// TIA Portal V17 export
// export: Created 2026-04-13T11:12:52.8832343Z, ExportSetting WithDefaults, DisplayName Totally Integrated Automation Portal, DisplayVersion V17 Update 4, DisplayName TIA Portal Openness, DisplayVersion V17 Update 4, DisplayName TIA Portal Version Control Interface, DisplayVersion V17, DisplayName SINAMICS Startdrive Advanced, DisplayVersion V17, DisplayName SINAMICS Startdrive G130, G150, S120, S150, SINAMICS MV, S210, DisplayVersion V17, DisplayName SINAMICS Startdrive G110M, G120, G120C, G120D, G120P, G115D, DisplayVersion V17, DisplayName STEP 7 Professional, DisplayVersion V17 Update 4, DisplayName STEP 7 Safety, DisplayVersion V17, DisplayName WinCC Professional, DisplayVersion V17 Update 4
TagTable "INCIP"
  INCIP_DD电导合格值 : Real  (PLC tag INCIP.DD电导合格值, HMI_连接_1, 1 s)
  INCIP_JX碱洗温度设定 : Real  (PLC tag INCIP.JX碱洗温度设定, HMI_连接_1, 1 s)
  INCIP_DD电导率当前值 : Real  (PLC tag INCIP.DD电导率当前值, HMI_连接_1, 1 s)
  INCIP_JX碱洗温度 : Real  (PLC tag INCIP.JX碱洗温度, HMI_连接_1, 1 s)
  INCIP_CIP压力 : Real  (PLC tag INCIP.CIP压力, HMI_连接_1, 1 s)
  INCIP_MZD自动清洗 : Bool  (PLC tag INCIP.MZD自动清洗, HMI_连接_1, 1 s)
  INCIP_MSD手动_纯水清洗 : Bool  (PLC tag INCIP.MSD手动_纯水清洗, HMI_连接_1, 1 s)
  INCIP_MSD手动_碱水清洗 : Bool  (PLC tag INCIP.MSD手动_碱水清洗, HMI_连接_1, 1 s)
  INCIP_MSD手动_溶剂清洗 : Bool  (PLC tag INCIP.MSD手动_溶剂清洗, HMI_连接_1, 1 s)
  INCIP_MSD手动_热水清洗 : Bool  (PLC tag INCIP.MSD手动_热水清洗, HMI_连接_1, 1 s)
  INCIP_MQX清洗重置 : Bool  (PLC tag INCIP.MQX清洗重置, HMI_连接_1, 1 s)
  INCIP_MCS纯水罐阀门 : Bool  (PLC tag INCIP.MCS纯水罐阀门, HMI_连接_1, 1 s)
  INCIP_MJS碱水罐阀门 : Bool  (PLC tag INCIP.MJS碱水罐阀门, HMI_连接_1, 1 s)
  INCIP_MZS注射水阀门 : Bool  (PLC tag INCIP.MZS注射水阀门, HMI_连接_1, 1 s)
  INCIP_MYK压空吹干阀 : Bool  (PLC tag INCIP.MYK压空吹干阀, HMI_连接_1, 1 s)
  INCIP_MD清洗失败 : Bool  (PLC tag INCIP.MD清洗失败, HMI_连接_1, 1 s)
  INCIP_MQX室内清洗辅助 : Bool  (PLC tag INCIP.MQX室内清洗辅助, HMI_连接_1, 1 s)
  INCIP_MZT主塔清洗头 : Bool  (PLC tag INCIP.MZT主塔清洗头, HMI_连接_1, 1 s)
  INCIP_MZT中途停止 : Bool  (PLC tag INCIP.MZT中途停止, HMI_连接_1, 1 s)
  INCIP_MXT心跳信号发送 : Bool  (PLC tag INCIP.MXT心跳信号发送, HMI_连接_1, 1 s)
  INCIP_MXT心跳信号接受 : Bool  (PLC tag INCIP.MXT心跳信号接受, HMI_连接_1, 1 s)
  INCIP_MXY泄压请求 : Bool  (PLC tag INCIP.MXY泄压请求, HMI_连接_1, 1 s)
  INCIP_MGS供水泵请求 : Bool  (PLC tag INCIP.MGS供水泵请求, HMI_连接_1, 1 s)
  INCIP_MCIP远程状态 : Bool  (PLC tag INCIP.MCIP远程状态, HMI_连接_1, 1 s)
  INCIP_QCS纯水罐阀门 : Bool  (PLC tag INCIP.QCS纯水罐阀门, HMI_连接_1, 1 s)
  INCIP_QJS碱水罐阀门 : Bool  (PLC tag INCIP.QJS碱水罐阀门, HMI_连接_1, 1 s)
  INCIP_QZS注射水罐阀门 : Bool  (PLC tag INCIP.QZS注射水罐阀门, HMI_连接_1, 1 s)
  INCIP_QYG压干阀门 : Bool  (PLC tag INCIP.QYG压干阀门, HMI_连接_1, 1 s)
  INCIP_QGS供水泵状态CIP : Bool  (PLC tag INCIP.QGS供水泵状态CIP, HMI_连接_1, 1 s)
  INCIP_QXY泄压阀门 : Bool  (PLC tag INCIP.QXY泄压阀门, HMI_连接_1, 1 s)
  INCIP_PS排水时间 : Real  (PLC tag INCIP.PS排水时间, HMI_连接_1, 1 s)
  INCIP_PS排水时间计时 : Real  (PLC tag INCIP.PS排水时间计时, HMI_连接_1, 1 s)
